TYPE ST_CreatedTime :
STRUCT
	isYearCreated : BIT;
	isMonthCreated : BIT;
	isDayCreated : BIT;
	isHourCreated : BIT;
	isMinuteCreated : BIT;
	isSecondCreated : BIT;
END_STRUCT
END_TYPE

(* stored: Version 1.1.0.1, ProductVersion 3.1.4024.12
   DUT ST_CreatedTime: Id {25fde252-3a1a-458c-a789-d5985df422e6} *)
